(* IEC 61131-3 sources: sntp/src/serialization/communication/BigEndian, 3 files *)

(* ---- LSNTP_typeTelegram.st ---- *)
// This is generated code. *** DO NOT MODIFY ***

NAMESPACE Simatic.Ax.sntp
FUNCTION SerializeBig : UDINT
    VAR_INPUT
        offset : UDINT;
    END_VAR
    VAR_IN_OUT
        value : LSNTP_typeTelegram;
        buffer : ARRAY[*] OF BYTE;
    END_VAR
    VAR_TEMP
        i : DINT;
    END_VAR
    SerializeBig := offset;
    FOR i := DINT#0 TO DINT#3 DO
        SerializeBig := System.Serialization.SerializeBig(offset := SerializeBig, value := value.flags[i], buffer := buffer);
    END_FOR;
    SerializeBig := System.Serialization.SerializeBig(offset := SerializeBig, value := value.rootDelay, buffer := buffer);
    SerializeBig := System.Serialization.SerializeBig(offset := SerializeBig, value := value.rootDispersion, buffer := buffer);
    FOR i := DINT#0 TO DINT#3 DO
        SerializeBig := System.Serialization.SerializeBig(offset := SerializeBig, value := value.referenceId[i], buffer := buffer);
    END_FOR;
    SerializeBig := SerializeBig(offset := SerializeBig, value := value.timestamps, buffer := buffer);
END_FUNCTION

FUNCTION DeserializeBig : UDINT
    VAR_INPUT
        offset : UDINT;
        buffer : ARRAY[*] OF BYTE;
    END_VAR
    VAR_IN_OUT
        value : LSNTP_typeTelegram;
    END_VAR
    VAR_TEMP
        i : DINT;
    END_VAR
    DeserializeBig := offset;
    FOR i := DINT#0 TO DINT#3 DO
        DeserializeBig := System.Serialization.DeserializeBig(offset := DeserializeBig, value := value.flags[i], buffer := buffer);
    END_FOR;
    DeserializeBig := System.Serialization.DeserializeBig(offset := DeserializeBig, value := value.rootDelay, buffer := buffer);
    DeserializeBig := System.Serialization.DeserializeBig(offset := DeserializeBig, value := value.rootDispersion, buffer := buffer);
    FOR i := DINT#0 TO DINT#3 DO
        DeserializeBig := System.Serialization.DeserializeBig(offset := DeserializeBig, value := value.referenceId[i], buffer := buffer);
    END_FOR;
    DeserializeBig := DeserializeBig(offset := DeserializeBig, value := value.timestamps, buffer := buffer);
END_FUNCTION
END_NAMESPACE

(* ---- LSNTP_typeTimestamp.st ---- *)
// This is generated code. *** DO NOT MODIFY ***

NAMESPACE Simatic.Ax.sntp
FUNCTION SerializeBig : UDINT
    VAR_INPUT
        offset : UDINT;
    END_VAR
    VAR_IN_OUT
        value : LSNTP_typeTimestamp;
        buffer : ARRAY[*] OF BYTE;
    END_VAR
    SerializeBig := offset;
    SerializeBig := System.Serialization.SerializeBig(offset := SerializeBig, value := value.sec, buffer := buffer);
    SerializeBig := System.Serialization.SerializeBig(offset := SerializeBig, value := value.secFrac, buffer := buffer);
END_FUNCTION

FUNCTION DeserializeBig : UDINT
    VAR_INPUT
        offset : UDINT;
        buffer : ARRAY[*] OF BYTE;
    END_VAR
    VAR_IN_OUT
        value : LSNTP_typeTimestamp;
    END_VAR
    DeserializeBig := offset;
    DeserializeBig := System.Serialization.DeserializeBig(offset := DeserializeBig, value := value.sec, buffer := buffer);
    DeserializeBig := System.Serialization.DeserializeBig(offset := DeserializeBig, value := value.secFrac, buffer := buffer);
END_FUNCTION
END_NAMESPACE

(* ---- LSNTP_typeTimestamps.st ---- *)
// This is generated code. *** DO NOT MODIFY ***

NAMESPACE Simatic.Ax.sntp
FUNCTION SerializeBig : UDINT
    VAR_INPUT
        offset : UDINT;
    END_VAR
    VAR_IN_OUT
        value : LSNTP_typeTimestamps;
        buffer : ARRAY[*] OF BYTE;
    END_VAR
    SerializeBig := offset;
    SerializeBig := SerializeBig(offset := SerializeBig, value := value.reference, buffer := buffer);
    SerializeBig := SerializeBig(offset := SerializeBig, value := value.originate, buffer := buffer);
    SerializeBig := SerializeBig(offset := SerializeBig, value := value.receive, buffer := buffer);
    SerializeBig := SerializeBig(offset := SerializeBig, value := value.transmit, buffer := buffer);
END_FUNCTION

FUNCTION DeserializeBig : UDINT
    VAR_INPUT
        offset : UDINT;
        buffer : ARRAY[*] OF BYTE;
    END_VAR
    VAR_IN_OUT
        value : LSNTP_typeTimestamps;
    END_VAR
    DeserializeBig := offset;
    DeserializeBig := DeserializeBig(offset := DeserializeBig, value := value.reference, buffer := buffer);
    DeserializeBig := DeserializeBig(offset := DeserializeBig, value := value.originate, buffer := buffer);
    DeserializeBig := DeserializeBig(offset := DeserializeBig, value := value.receive, buffer := buffer);
    DeserializeBig := DeserializeBig(offset := DeserializeBig, value := value.transmit, buffer := buffer);
END_FUNCTION
END_NAMESPACE
